PROGRAM MAIN
VAR
	mcMover						: ARRAY [1..ciMoverMax] OF MC_PlanarMover;
	i							: INT;
END_VAR
VAR
	CONSTANT
	ciMoverMax					: INT := 4;
END_VAR

FOR i:= 1 TO ciMoverMax DO
	mcMover[i].Update();
END_FOR

END_PROGRAM

(* stored: Version 1.1.0.1, ProductVersion 3.1.4024.12
   POU MAIN: Id {058cc226-bb0f-4c5e-b6c5-adf46d7b7173}, SpecialFunc None *)
